(*
	This structure contains all the outputs of the BANNER LED.
	The inputs and the outputs are linked to the device as well.
*)
TYPE ST_Banner_K30PTKQ_Status :
	STRUCT
	OutputState	: UINT; (* 0 = Normally Closed, 1 = Normally Open *)
	END_STRUCT
END_TYPE

(* stored: Version 1.1.0.1, ProductVersion 3.1.4024.12
   DUT ST_Banner_K30PTKQ_Status: Id {c86f365a-7409-44ba-9973-3350ac137dbd} *)
